// SIMATIC S7-200 project (STEP 7-Micro/WIN), CPU 224 REL 02.01

SYMBOL_TABLE Modbus Protocol (v1.0)
ModbusBufr       VB0      // Dirección de un búfer de 256 bytes
END_SYMBOL_TABLE

ORGANIZATION_BLOCK PRINCIPAL:OB1
TITLE=COMENTARIOS DEL PROGRAMA
BEGIN
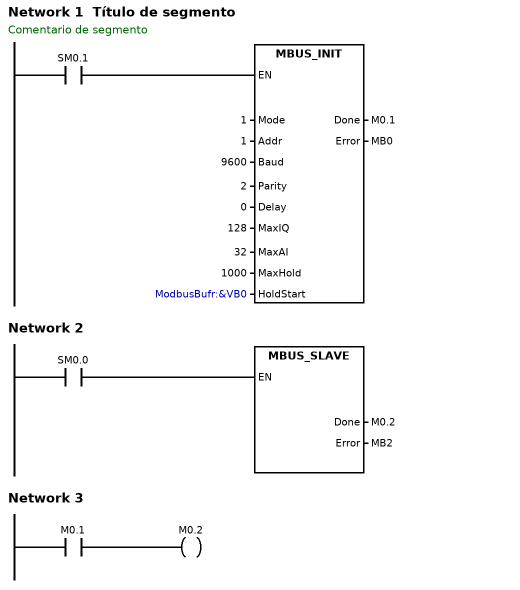
Network 1 // Título de segmento
// Comentario de segmento
LD     SM0.1
CALL   MBUS_INIT:SBR1, 1, 1, 9600, 2, 0, 128, 32, 1000, &ModbusBufr:VB0, M0.1, MB0
Network 2
LD     SM0.0
CALL   MBUS_SLAVE:SBR2, M0.2, MB2
Network 3
LD     M0.1
=      M0.2
END_ORGANIZATION_BLOCK

// SBR1: protected block, not included

// SBR2: protected block, not included

// SBR3: protected block, not included
